// TIA Portal V20 export
TYPE "LKinCtrl_PointEditor_typeInternalEvents"
// stored: Access Published
   STRUCT
      touchUp { ExternalAccessible := 'False'; ExternalVisible := 'False'; ExternalWritable := 'False'} : Struct
         trigger : Bool;
         index : DInt;   // Index in point table. -1: currently selected point
         keepName : Bool;
         point : "LKinCtrl_typePoint";   // New point
      END_STRUCT;
   END_STRUCT;
END_TYPE
